FUNCTION_BLOCK fbVacuumValveCtrl

VAR_INPUT
	IN_Name:				STRING;
	In_Enable:				BOOL;
	In_Reset:				BOOL;


	(*Sensors*)
	In_Vacuum_Switch:		BOOL;
	In_Drop_Monitor_Enable:	BOOL;

	(*Timer*)
	In_VacuumTON:			TIME;
	In_Release_TON:			TIME;
	In_PurgeTON:			TIME;
	in_Timeout:				TIME;
END_VAR

VAR_OUTPUT
	Out_VacuumSV:			BOOL;
	Out_PurgeSV:			BOOL;
END_VAR

VAR

	Loc_Vacuum:				BOOL;
	Loc_Purge:				BOOL;
	Err_Vacuum:				BOOL;
	VAcuum_TOut:			TON;
	Purge_TOut: 				TON;
	Vacuum_TON:			TON;
	Release_TON: 			TON;
	Purge_TON:				TON;
	Purge_ON:				BOOL;
	Loc_VacuumPls: 			BOOL;
	PurgePls:				R_TRIG;
	VacuumPls: 				R_TRIG;
	Loc_PurgePls: 			BOOL;
	Out_RSErr:				BOOL;
	VacuumPosPls: 			F_TRIG;
	PurgePosPls: 			F_TRIG;
	plsManualOff: R_TRIG;
END_VAR
VAR_IN_OUT
	VacVar:structVacuum;
	Station:structStationCtrl;
END_VAR
VAR // added by the converter: edge detectors and wires of the graphical bodies
    _w1, _w2, _w3, _w4, _w5 : BOOL;
END_VAR

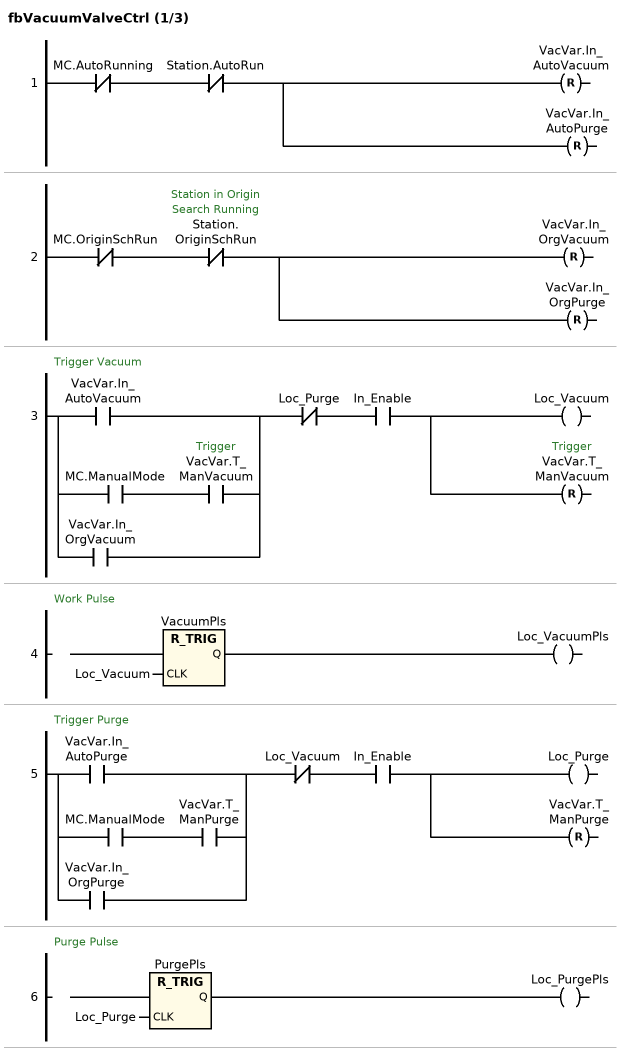
// NETWORK 1
_w1 := NOT MC.AutoRunning AND NOT Station.AutoRun;
VacVar.In_AutoVacuum R= _w1;
VacVar.In_AutoPurge R= _w1;

// NETWORK 2
//   Station.OriginSchRun: Station in Origin Search Running
_w2 := NOT MC.OriginSchRun AND NOT Station.OriginSchRun;
VacVar.In_OrgVacuum R= _w2;
VacVar.In_OrgPurge R= _w2;

// NETWORK 3
// Trigger Vacuum
//   VacVar.T_ManVacuum: Trigger
_w3 := (VacVar.In_AutoVacuum OR MC.ManualMode AND VacVar.T_ManVacuum OR VacVar.In_OrgVacuum) AND NOT Loc_Purge AND In_Enable;
Loc_Vacuum := _w3;
VacVar.T_ManVacuum R= _w3;

// NETWORK 4
// Work Pulse
VacuumPls(CLK := Loc_Vacuum); // R_TRIG
Loc_VacuumPls := VacuumPls.Q;

// NETWORK 5
// Trigger Purge
_w4 := (VacVar.In_AutoPurge OR MC.ManualMode AND VacVar.T_ManPurge OR VacVar.In_OrgPurge) AND NOT Loc_Vacuum AND In_Enable;
Loc_Purge := _w4;
VacVar.T_ManPurge R= _w4;

// NETWORK 6
// Purge Pulse
PurgePls(CLK := Loc_Purge); // R_TRIG
Loc_PurgePls := PurgePls.Q;

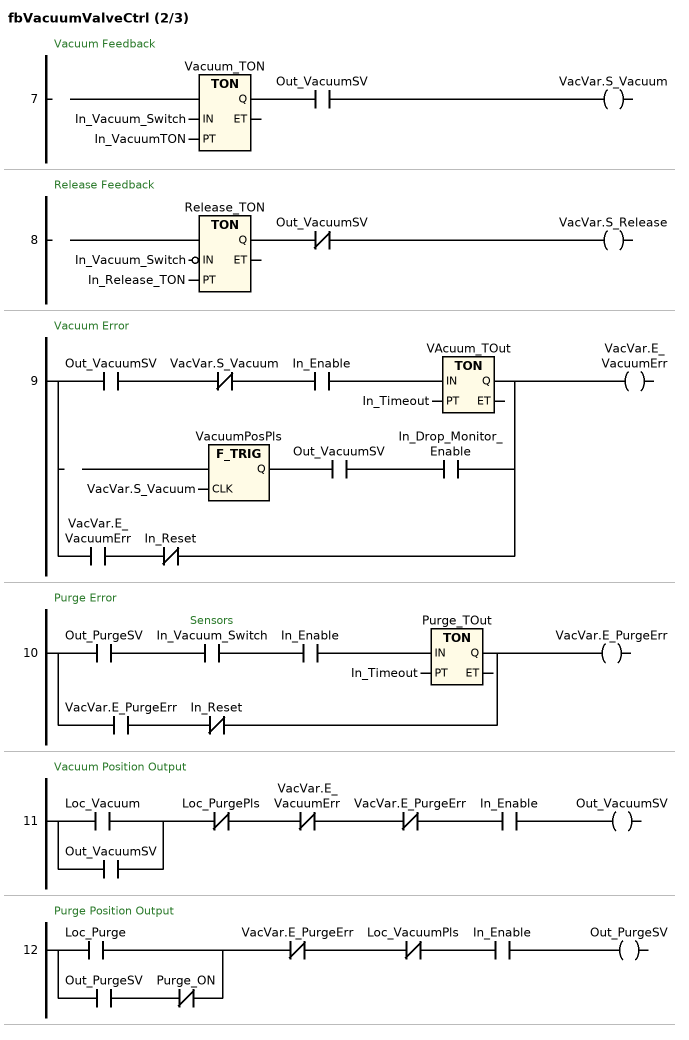
// NETWORK 7
// Vacuum Feedback
//   In_Vacuum_Switch: Sensors
//   In_VacuumTON: Timer
Vacuum_TON(IN := In_Vacuum_Switch, PT := In_VacuumTON); // TON
VacVar.S_Vacuum := Vacuum_TON.Q AND Out_VacuumSV;

// NETWORK 8
// Release Feedback
//   In_Vacuum_Switch: Sensors
Release_TON(IN := NOT In_Vacuum_Switch, PT := In_Release_TON); // TON
VacVar.S_Release := Release_TON.Q AND NOT Out_VacuumSV;

// NETWORK 9
// Vacuum Error
VAcuum_TOut(IN := Out_VacuumSV AND NOT VacVar.S_Vacuum AND In_Enable, PT := In_Timeout); // TON
VacuumPosPls(CLK := VacVar.S_Vacuum); // F_TRIG
VacVar.E_VacuumErr := VAcuum_TOut.Q OR VacuumPosPls.Q AND Out_VacuumSV AND In_Drop_Monitor_Enable OR VacVar.E_VacuumErr AND NOT In_Reset;

// NETWORK 10
// Purge Error
//   In_Vacuum_Switch: Sensors
Purge_TOut(IN := Out_PurgeSV AND In_Vacuum_Switch AND In_Enable, PT := In_Timeout); // TON
VacVar.E_PurgeErr := Purge_TOut.Q OR VacVar.E_PurgeErr AND NOT In_Reset;

// NETWORK 11
// Vacuum Position Output
Out_VacuumSV := (Loc_Vacuum OR Out_VacuumSV) AND NOT Loc_PurgePls AND NOT VacVar.E_VacuumErr AND NOT VacVar.E_PurgeErr AND In_Enable;

// NETWORK 12
// Purge Position Output
Out_PurgeSV := (Loc_Purge OR Out_PurgeSV AND NOT Purge_ON) AND NOT VacVar.E_PurgeErr AND NOT Loc_VacuumPls AND In_Enable;

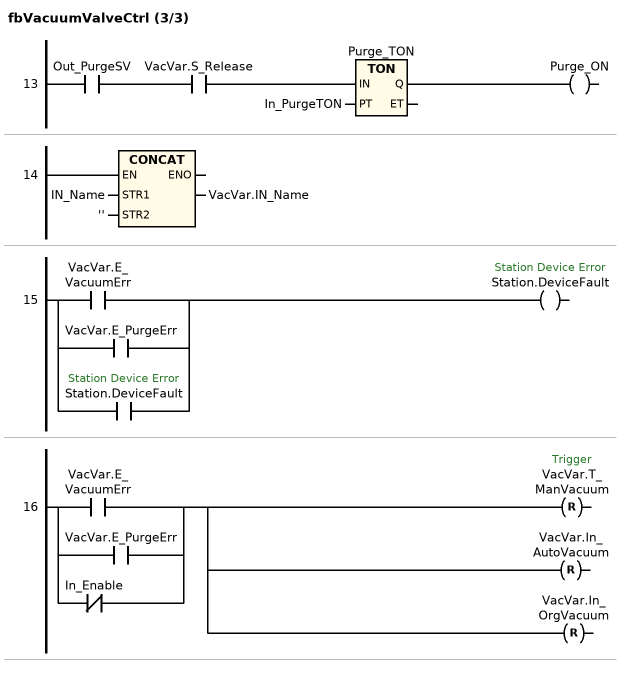
// NETWORK 13
Purge_TON(IN := Out_PurgeSV AND VacVar.S_Release, PT := In_PurgeTON); // TON
Purge_ON := Purge_TON.Q;

// NETWORK 14
VacVar.IN_Name := CONCAT(STR1 := IN_Name, STR2 := '');

// NETWORK 15
//   Station.DeviceFault: Station Device Error
Station.DeviceFault := VacVar.E_VacuumErr OR VacVar.E_PurgeErr OR Station.DeviceFault;

// NETWORK 16
//   VacVar.T_ManVacuum: Trigger
_w5 := VacVar.E_VacuumErr OR VacVar.E_PurgeErr OR NOT In_Enable;
VacVar.T_ManVacuum R= _w5;
VacVar.In_AutoVacuum R= _w5;
VacVar.In_OrgVacuum R= _w5;

END_FUNCTION_BLOCK

(* stored: Version 1.1.0.1, ProductVersion 3.1.4018.2
   POU fbVacuumValveCtrl: Id {ce946103-2a0f-4d3d-9696-305bd245a28d}, SpecialFunc None *)
